PROGRAM MAIN
VAR
END_VAR

CASE GVL.nProgramID OF
	0 : Reset();
	1 : V0_1();
	2 : V0_2();
	3 : V0_3();
END_CASE

END_PROGRAM

(* stored: Version 1.1.0.1, ProductVersion 3.1.4024.12
   POU MAIN: Id {802f884d-54f5-444a-9d44-2eadbfbf0423}, SpecialFunc None *)
